(* IEC 61131-3 sources: beckhoffAutomationInterface/ST/Shark/Lib/BehaviorTree/actions, 12 files *)

(* ---- FB_AlwaysFailureNode.st ---- *)
FUNCTION_BLOCK FB_AlwaysFailureNode IMPLEMENTS I_TreeNode
VAR_INPUT
    sName : STRING(50) := 'Always Failure';
END_VAR

METHOD Tick : ST_NodeResult
    Tick.eStatus := E_NodeStatus.FAILURE;
    Tick.bHasError := TRUE;
    Tick.stError.eErrorId := E_ErrorId.ERR_BT_FORCED_FAILURE;
    Tick.stError.sSource := sName;
    Tick.stError.sMessage := 'Forced Failure';
    Tick.sDescription := CONCAT(sName, ' - Failure');
END_METHOD

{attribute 'estimated-stack-usage' := '500'}
METHOD Reset : BOOL
    Reset := TRUE;
END_METHOD

{attribute 'estimated-stack-usage' := '500'}
METHOD Halt
END_METHOD
END_FUNCTION_BLOCK

(* ---- FB_AlwaysSuccessNode.st ---- *)
FUNCTION_BLOCK FB_AlwaysSuccessNode IMPLEMENTS I_TreeNode
VAR_INPUT
    sName : STRING(50) := 'Always Success';
END_VAR

METHOD Tick : ST_NodeResult
    Tick.eStatus := E_NodeStatus.SUCCESS;
    Tick.rProgress := 100.0;
    Tick.sDescription := CONCAT(sName, ' - Success');
END_METHOD

{attribute 'estimated-stack-usage' := '500'}
METHOD Reset : BOOL
    Reset := TRUE;
END_METHOD

{attribute 'estimated-stack-usage' := '500'}
METHOD Halt
END_METHOD
END_FUNCTION_BLOCK

(* ---- FB_CheckSensorNode.st ---- *)
FUNCTION_BLOCK FB_CheckSensorNode IMPLEMENTS I_TreeNode
VAR_INPUT
    sName : STRING(50) := 'Check Sensor Node';
END_VAR
VAR
    _ipSensor     : I_Sensor;
    _rThreshold   : LREAL;
    _eCompareMode : E_CompareMode := E_CompareMode.GREATER_THAN;
    _rTolerance   : LREAL;
    _rLastValue   : LREAL;
END_VAR

METHOD PUBLIC Init : BOOL
VAR_INPUT
    ipSensor   : I_Sensor;
    rThreshold : LREAL;
    eMode      : E_CompareMode := E_CompareMode.GREATER_THAN;
    rTolerance : LREAL := 0.0;
    sNodeName  : STRING(50) := '';
END_VAR
    IF ipSensor = 0 THEN RETURN; END_IF
    _ipSensor     := ipSensor;
    _rThreshold   := rThreshold;
    _eCompareMode := eMode;
    _rTolerance   := rTolerance;
    IF sNodeName <> '' THEN sName := sNodeName; END_IF
    Init := TRUE;
END_METHOD

PROPERTY PUBLIC Threshold : LREAL
    GET
    Threshold := _rThreshold;
    END_GET
    SET
    _rThreshold := Threshold;
    END_SET
END_PROPERTY

PROPERTY PUBLIC CompareMode : E_CompareMode
    GET
    CompareMode := _eCompareMode;
    END_GET
    SET
    _eCompareMode := CompareMode;
    END_SET
END_PROPERTY

METHOD PRIVATE GetStatusDescription : STRING(255)
VAR
    sResult : STRING(255);
END_VAR
    sResult := CONCAT(sName, ' - current=');
    sResult := CONCAT(sResult, LREAL_TO_FMTSTR(_rLastValue, 2, TRUE));
    sResult := CONCAT(sResult, CONCAT(', threshold=', LREAL_TO_FMTSTR(_rThreshold, 2, TRUE)));
    IF _eCompareMode = E_CompareMode.WITHIN_TOLERANCE AND _rTolerance > 0.0 THEN
        sResult := CONCAT(sResult, CONCAT(' +/-', LREAL_TO_FMTSTR(_rTolerance, 2, TRUE)));
    ELSE
        sResult := CONCAT(sResult, CONCAT(' (', CONCAT(F_CompareModeToString(_eCompareMode), ')')));
    END_IF
    GetStatusDescription := sResult;
END_METHOD

METHOD Tick : ST_NodeResult
VAR
    rCurrent  : LREAL;
    sErrorMsg : STRING(255);
END_VAR
    IF _ipSensor = 0 THEN
        Tick := F_BuildNullInterfaceResult(sName, 'Sensor interface not configured');
        RETURN;
    END_IF

    IF _ipSensor.IsError() THEN
        Tick.eStatus := E_NodeStatus.FAILURE;
        Tick.bHasError := TRUE;
        Tick.stError.eErrorId := E_ErrorId.ERR_BT_SENSOR_ERROR;
        Tick.stError.sSource := sName;
        Tick.stError.sMessage := 'Sensor reported error';
        RETURN;
    END_IF

    rCurrent    := _ipSensor.GetMeasurement();
    _rLastValue := rCurrent;

    IF F_EvaluateCompareMode(rCurrent, _rThreshold, _rTolerance, _eCompareMode) THEN
        Tick.eStatus := E_NodeStatus.SUCCESS;
        Tick.rProgress := 100.0;
        Tick.sDescription := GetStatusDescription();
    ELSE
        sErrorMsg := CONCAT('Value ', LREAL_TO_FMTSTR(rCurrent, 2, TRUE));
        sErrorMsg := CONCAT(sErrorMsg, CONCAT(' not ', F_CompareModeToString(_eCompareMode)));
        sErrorMsg := CONCAT(sErrorMsg, CONCAT(' ', LREAL_TO_FMTSTR(_rThreshold, 2, TRUE)));

        Tick.eStatus := E_NodeStatus.FAILURE;
        Tick.bHasError := TRUE;
        Tick.stError.eErrorId := E_ErrorId.ERR_BT_CONDITION_FAILED;
        Tick.stError.sSource := sName;
        Tick.stError.sMessage := sErrorMsg;
        Tick.sDescription := GetStatusDescription();
    END_IF
END_METHOD

{attribute 'estimated-stack-usage' := '500'}
METHOD Halt
    // No explicit action required
END_METHOD

{attribute 'estimated-stack-usage' := '500'}
METHOD Reset : BOOL
    Reset := TRUE;
END_METHOD

END_FUNCTION_BLOCK

(* ---- FB_CloseValveNode.st ---- *)
FUNCTION_BLOCK FB_CloseValveNode IMPLEMENTS I_TreeNode
VAR_INPUT
    sName : STRING(50) := 'Close Valve';
END_VAR
VAR
    _ipValve : I_Valve;
END_VAR

METHOD PUBLIC Init : BOOL
VAR_INPUT
    ipValve   : I_Valve;
    sNodeName : STRING(50) := '';
END_VAR
    IF ipValve = 0 THEN RETURN; END_IF
    _ipValve := ipValve;
    IF sNodeName <> '' THEN sName := sNodeName; END_IF
    Init := TRUE;
END_METHOD

METHOD Tick : ST_NodeResult
VAR
    stValveError : ST_Error;
END_VAR
    IF _ipValve = 0 THEN
        Tick := F_BuildNullInterfaceResult(sName, 'Valve interface not configured');
        RETURN;
    END_IF

    _ipValve.Close();

    IF _ipValve.IsClosed() THEN
        Tick.eStatus := E_NodeStatus.SUCCESS;
        Tick.rProgress := 100.0;
        Tick.sDescription := CONCAT(sName, ' - Valve closed');
    ELSIF _ipValve.IsError() THEN
        stValveError := _ipValve.GetError();
        Tick.eStatus := E_NodeStatus.FAILURE;
        Tick.bHasError := TRUE;
        Tick.stError.sSource := sName;

        IF stValveError.eErrorId <> E_ErrorId.NO_ERROR THEN
            Tick.stError.eErrorId := stValveError.eErrorId;
            Tick.stError.sMessage := stValveError.sMessage;
        ELSE
            Tick.stError.eErrorId := E_ErrorId.ERR_BT_VALVE_ERROR;
            Tick.stError.sMessage := 'Valve reported error while closing';
        END_IF
    ELSE
        Tick.eStatus := E_NodeStatus.RUNNING;
        Tick.sDescription := CONCAT(sName, ' - Closing valve, currently open');
    END_IF
END_METHOD

{attribute 'estimated-stack-usage' := '500'}
METHOD Reset : BOOL
    Reset := TRUE;
END_METHOD

{attribute 'estimated-stack-usage' := '500'}
METHOD Halt
    // Safe state: ensure the valve is closed (isolated).
    IF _ipValve <> 0 THEN
        _ipValve.Close();
    END_IF
END_METHOD

END_FUNCTION_BLOCK

(* ---- FB_ConditionNode.st ---- *)
// FB_ConditionNode - Pure leaf node that evaluates a boolean condition
// Returns SUCCESS if condition is TRUE, FAILURE if FALSE
// This is a leaf node, it has no child.
//
// Usage:
//   fbCondition.Init(refCondition := bMyFlag);
//   fbSequence.AddChild(fbCondition);
//
FUNCTION_BLOCK FB_ConditionNode IMPLEMENTS I_TreeNode
VAR_INPUT
    sName : STRING(50) := 'Condition Node';
END_VAR
VAR
    _refCondition : REFERENCE TO BOOL;
    _bInvertResult : BOOL := FALSE;
END_VAR

    // Configure with reference to boolean condition
METHOD PUBLIC Init : BOOL
VAR_INPUT
    refCondition  : REFERENCE TO BOOL;
    bInvertResult : BOOL := FALSE; // Optional: invert the result
    sNodeName     : STRING(50) := '';
END_VAR
    IF NOT __ISVALIDREF(refCondition) THEN
        Init := FALSE;
        RETURN;
    END_IF

    _refCondition REF= refCondition;
    _bInvertResult := bInvertResult;
    IF sNodeName <> '' THEN sName := sNodeName; END_IF
    Init := TRUE;
END_METHOD

METHOD Tick : ST_NodeResult
VAR
    bConditionValue : BOOL;
END_VAR

    IF NOT __ISVALIDREF(_refCondition) THEN
        Tick.eStatus := E_NodeStatus.FAILURE;
        Tick.bHasError := TRUE;
        Tick.stError.eErrorId := E_ErrorId.ERR_BT_CONDITION_NOT_CONFIGURED;
        Tick.stError.sSource := sName;
        Tick.stError.sMessage := 'Condition reference not configured';
        RETURN;
    END_IF

    bConditionValue := _refCondition;

    // Apply inversion if configured
    IF _bInvertResult THEN
        bConditionValue := NOT bConditionValue;
    END_IF

    IF bConditionValue THEN
        Tick.eStatus := E_NodeStatus.SUCCESS;
        Tick.sDescription := CONCAT(sName, ' - Condition Met');
        Tick.rProgress := 100.0;
    ELSE
        // Condition false is not an error - it's expected behavior
        Tick.eStatus := E_NodeStatus.FAILURE;
        Tick.sDescription := CONCAT(sName, ' - Condition Not Met');
    END_IF
END_METHOD

{attribute 'estimated-stack-usage' := '500'}
METHOD Halt
    // Nothing to halt
END_METHOD

{attribute 'estimated-stack-usage' := '500'}
METHOD Reset : BOOL
    Reset := TRUE;
END_METHOD

END_FUNCTION_BLOCK

(* ---- FB_EnableControllerNode.st ---- *)
FUNCTION_BLOCK FB_EnableControllerNode IMPLEMENTS I_TreeNode
VAR_INPUT
    sName : STRING(50) := 'Enable Controller';
END_VAR
VAR
    _ipController : I_Controller;
    _bEnable      : BOOL;
END_VAR

METHOD PUBLIC Init : BOOL
VAR_INPUT
    ipController : I_Controller;
    bEnable      : BOOL;
    sNodeName    : STRING(50) := '';
END_VAR
    IF ipController = 0 THEN RETURN; END_IF
    _ipController := ipController;
    _bEnable      := bEnable;
    IF sNodeName <> '' THEN sName := sNodeName; END_IF
    Init := TRUE;
END_METHOD

METHOD Tick : ST_NodeResult
    IF _ipController = 0 THEN
        Tick := F_BuildNullInterfaceResult(sName, 'Controller interface not configured');
        RETURN;
    END_IF

    _ipController.Enable(_bEnable);
    Tick.eStatus := E_NodeStatus.SUCCESS;
    Tick.rProgress := 100.0;
    IF _bEnable THEN
        Tick.sDescription := CONCAT(sName, ' - Enabling controller');
    ELSE
        Tick.sDescription := CONCAT(sName, ' - Disabling controller');
    END_IF
END_METHOD

{attribute 'estimated-stack-usage' := '500'}
METHOD Reset : BOOL
    Reset := TRUE;
END_METHOD

{attribute 'estimated-stack-usage' := '500'}
METHOD Halt
    // Safe state: disable the controller.
    IF _ipController <> 0 THEN
        _ipController.Enable(FALSE);
    END_IF
END_METHOD

END_FUNCTION_BLOCK

(* ---- FB_MonitorControllerNode.st ---- *)
(* FB_MonitorControllerNode - Monitor controller for errors while running

BEHAVIOR:
- Returns RUNNING while controller has no error
- Returns FAILURE immediately if controller reports error
- Never returns SUCCESS on its own (used in parallel with other nodes)

USE CASE:
Run in parallel with other nodes. If the controller enters an error state
this node fails immediately, causing the parallel node to fail without
waiting for the other branches to complete.
*)
FUNCTION_BLOCK FB_MonitorControllerNode IMPLEMENTS I_TreeNode
VAR_INPUT
    sName : STRING(50) := 'Monitor Controller Node';
END_VAR
VAR
    _ipController : I_Controller;
END_VAR

METHOD PUBLIC Init : BOOL
VAR_INPUT
    ipController : I_Controller;
    sNodeName    : STRING(50) := '';
END_VAR
    IF ipController = 0 THEN RETURN; END_IF
    _ipController := ipController;
    IF sNodeName <> '' THEN sName := sNodeName; END_IF
    Init := TRUE;
END_METHOD

METHOD Tick : ST_NodeResult
VAR
    stStatus : ST_ControllerStatus;
END_VAR
    IF _ipController = 0 THEN
        Tick := F_BuildNullInterfaceResult(sName, 'Controller interface not configured');
        RETURN;
    END_IF

    stStatus := _ipController.GetStatus();
    IF stStatus.stError.eErrorId <> E_ErrorId.NO_ERROR THEN
        Tick.eStatus := E_NodeStatus.FAILURE;
        Tick.bHasError := TRUE;
        Tick.stError := stStatus.stError;
        RETURN;
    END_IF

    Tick.eStatus := E_NodeStatus.RUNNING;
    Tick.sDescription := CONCAT(sName, ' - Monitoring (OK)');
END_METHOD

{attribute 'estimated-stack-usage' := '500'}
METHOD Halt
    // No explicit action required
END_METHOD

{attribute 'estimated-stack-usage' := '500'}
METHOD Reset : BOOL
    Reset := TRUE;
END_METHOD

END_FUNCTION_BLOCK

(* ---- FB_OpenValveNode.st ---- *)
FUNCTION_BLOCK FB_OpenValveNode IMPLEMENTS I_TreeNode
VAR_INPUT
    sName : STRING(50) := 'Open Valve';
END_VAR
VAR
    _ipValve : I_Valve;
END_VAR

METHOD PUBLIC Init : BOOL
VAR_INPUT
    ipValve   : I_Valve;
    sNodeName : STRING(50) := '';
END_VAR
    IF ipValve = 0 THEN RETURN; END_IF
    _ipValve := ipValve;
    IF sNodeName <> '' THEN sName := sNodeName; END_IF
    Init := TRUE;
END_METHOD

METHOD Tick : ST_NodeResult
VAR
    stValveError : ST_Error;
END_VAR
    IF _ipValve = 0 THEN
        Tick := F_BuildNullInterfaceResult(sName, 'Valve interface not configured');
        RETURN;
    END_IF

    _ipValve.Open();

    IF _ipValve.IsOpen() THEN
        Tick.eStatus := E_NodeStatus.SUCCESS;
        Tick.rProgress := 100.0;
        Tick.sDescription := CONCAT(sName, ' - Valve open');
    ELSIF _ipValve.IsError() THEN
        stValveError := _ipValve.GetError();
        Tick.eStatus := E_NodeStatus.FAILURE;
        Tick.bHasError := TRUE;
        Tick.stError.sSource := sName;

        IF stValveError.eErrorId <> E_ErrorId.NO_ERROR THEN
            Tick.stError.eErrorId := stValveError.eErrorId;
            Tick.stError.sMessage := stValveError.sMessage;
        ELSE
            Tick.stError.eErrorId := E_ErrorId.ERR_BT_VALVE_ERROR;
            Tick.stError.sMessage := 'Valve reported error while opening';
        END_IF
    ELSE
        Tick.eStatus := E_NodeStatus.RUNNING;
        Tick.sDescription := CONCAT(sName, ' - Opening valve, currently closed');
    END_IF
END_METHOD

{attribute 'estimated-stack-usage' := '500'}
METHOD Reset : BOOL
    Reset := TRUE;
END_METHOD

{attribute 'estimated-stack-usage' := '500'}
METHOD Halt
    // Safe state: isolate by closing the valve (SEQUENCE_BT_LIFECYCLE.md §3).
    IF _ipValve <> 0 THEN
        _ipValve.Close();
    END_IF
END_METHOD

END_FUNCTION_BLOCK

(* ---- FB_SetControllerNode.st ---- *)
FUNCTION_BLOCK FB_SetControllerNode IMPLEMENTS I_TreeNode
VAR_INPUT
    sName : STRING(50) := 'Set Controller';
END_VAR
VAR
    _ipController : I_Controller;
    _rSetpoint    : LREAL;
END_VAR

METHOD PUBLIC Init : BOOL
VAR_INPUT
    ipController : I_Controller;
    rSetpoint    : LREAL;
    sNodeName    : STRING(50) := '';
END_VAR
    IF ipController = 0 THEN RETURN; END_IF
    _ipController := ipController;
    _rSetpoint    := rSetpoint;
    IF sNodeName <> '' THEN sName := sNodeName; END_IF
    Init := TRUE;
END_METHOD

PROPERTY PUBLIC Setpoint : LREAL
    GET
    Setpoint := _rSetpoint;
    END_GET
    SET
    _rSetpoint := Setpoint;
    END_SET
END_PROPERTY

METHOD Tick : ST_NodeResult
    IF _ipController = 0 THEN
        Tick := F_BuildNullInterfaceResult(sName, 'Controller interface not configured');
        RETURN;
    END_IF

    _ipController.SetSetpoint(_rSetpoint);
    Tick.eStatus := E_NodeStatus.SUCCESS;
    Tick.rProgress := 100.0;
    Tick.sDescription := CONCAT(sName, CONCAT(' - Set setpoint=', LREAL_TO_FMTSTR(_rSetpoint, 2, TRUE)));
END_METHOD

{attribute 'estimated-stack-usage' := '500'}
METHOD Reset : BOOL
    Reset := TRUE;
END_METHOD

{attribute 'estimated-stack-usage' := '500'}
METHOD Halt
    // Safe state: zero the setpoint.
    IF _ipController <> 0 THEN
        _ipController.SetSetpoint(0.0);
    END_IF
END_METHOD

END_FUNCTION_BLOCK

(* ---- FB_SetDigitalOutputNode.st ---- *)
FUNCTION_BLOCK FB_SetDigitalOutputNode IMPLEMENTS I_TreeNode
VAR_INPUT
    sName : STRING(50) := 'Set Digital Output Node';
END_VAR
VAR
    _ipDO : I_DigitalOutput;
    _bState : BOOL;
END_VAR

METHOD PUBLIC Init : BOOL
VAR_INPUT
    ipDO      : I_DigitalOutput;
    bState    : BOOL;
    sNodeName : STRING(50) := '';
END_VAR
    IF ipDO = 0 THEN RETURN; END_IF
    _ipDO   := ipDO;
    _bState := bState;
    IF sNodeName <> '' THEN sName := sNodeName; END_IF
    Init := TRUE;
END_METHOD

METHOD Tick : ST_NodeResult
    IF _ipDO = 0 THEN
        Tick := F_BuildNullInterfaceResult(sName, 'Digital output interface not configured');
        RETURN;
    END_IF

    _ipDO.SetOutput(_bState);
    Tick.eStatus := E_NodeStatus.SUCCESS;
    Tick.sDescription := CONCAT(sName, ' - Output set');
    Tick.rProgress := 100.0;
END_METHOD

{attribute 'estimated-stack-usage' := '500'}
METHOD Halt
    // Apply the safe state configured at Init time.
    // The node has no knowledge of whether safe means TRUE or FALSE.
    IF _ipDO <> 0 THEN
        _ipDO.SetSafeState();
    END_IF
END_METHOD

{attribute 'estimated-stack-usage' := '500'}
METHOD Reset : BOOL
    Reset := TRUE;
END_METHOD

END_FUNCTION_BLOCK

(* ---- FB_WaitForSensorNode.st ---- *)
(* FB_WaitForSensorNode - Wait until sensor meets a condition

BEHAVIOR:
- Returns RUNNING while waiting for condition
- Returns SUCCESS when condition is met
- Returns FAILURE on errors (null sensor, sensor error) or timeout

TIMEOUT:
- tTimeout = T#0S  => no timeout, wait indefinitely (default)
- tTimeout > T#0S  => FAILURE with descriptive message when timeout expires

COMPARE MODES:
- WITHIN_TOLERANCE: ABS(value - target) <= tolerance (default)
- GREATER_THAN:     value > target
- LESS_THAN:        value < target
*)
FUNCTION_BLOCK FB_WaitForSensorNode IMPLEMENTS I_TreeNode
VAR_INPUT
    sName : STRING(50) := 'Wait For Sensor Node';
END_VAR
VAR
    _ipSensor     : I_Sensor;
    _rTarget      : LREAL;
    _rTolerance   : LREAL;
    _eCompareMode : E_CompareMode := E_CompareMode.WITHIN_TOLERANCE;
    _rLastValue   : LREAL;
    _tTimeout     : TIME := T#0S;
    _fbTimer      : TON;
    _bStarted     : BOOL;
END_VAR

METHOD PUBLIC Init : BOOL
VAR_INPUT
    ipSensor   : I_Sensor;
    rTarget    : LREAL;
    rTolerance : LREAL := 0.0;
    eMode      : E_CompareMode := E_CompareMode.WITHIN_TOLERANCE;
    tTimeout   : TIME := T#0S;
    sNodeName  : STRING(50) := '';
END_VAR
    IF ipSensor = 0 THEN RETURN; END_IF
    _ipSensor     := ipSensor;
    _rTarget      := rTarget;
    _rTolerance   := rTolerance;
    _eCompareMode := eMode;
    _tTimeout     := tTimeout;
    IF sNodeName <> '' THEN sName := sNodeName; END_IF
    Init := TRUE;
END_METHOD

PROPERTY PUBLIC Target : LREAL
    GET
    Target := _rTarget;
    END_GET
    SET
    _rTarget := Target;
    END_SET
END_PROPERTY

PROPERTY PUBLIC Tolerance : LREAL
    GET
    Tolerance := _rTolerance;
    END_GET
    SET
    _rTolerance := Tolerance;
    END_SET
END_PROPERTY

PROPERTY PUBLIC CompareMode : E_CompareMode
    GET
    CompareMode := _eCompareMode;
    END_GET
    SET
    _eCompareMode := CompareMode;
    END_SET
END_PROPERTY

PROPERTY PUBLIC Timeout : TIME
    GET
    Timeout := _tTimeout;
    END_GET
    SET
    _tTimeout := Timeout;
    END_SET
END_PROPERTY

METHOD PUBLIC GetStatusDescription : STRING(255)
VAR
    sResult : STRING(255);
END_VAR
    sResult := CONCAT(sName, ' - current=');
    sResult := CONCAT(sResult, LREAL_TO_FMTSTR(_rLastValue, 2, TRUE));
    sResult := CONCAT(sResult, CONCAT(', target=', LREAL_TO_FMTSTR(_rTarget, 2, TRUE)));
    IF _eCompareMode = E_CompareMode.WITHIN_TOLERANCE AND _rTolerance > 0.0 THEN
        sResult := CONCAT(sResult, CONCAT(' +/-', LREAL_TO_FMTSTR(_rTolerance, 2, TRUE)));
    ELSE
        sResult := CONCAT(sResult, CONCAT(' (', CONCAT(F_CompareModeToString(_eCompareMode), ')')));
    END_IF
    IF _tTimeout > T#0S AND _bStarted THEN
        sResult := CONCAT(sResult, CONCAT(' timeout=', CONCAT(TIME_TO_STRING(_fbTimer.ET), CONCAT('/', TIME_TO_STRING(_tTimeout)))));
    END_IF
    GetStatusDescription := sResult;
END_METHOD

METHOD Tick : ST_NodeResult
VAR
    rCurrentVal : LREAL;
END_VAR
    IF _ipSensor = 0 THEN
        Tick := F_BuildNullInterfaceResult(sName, 'Sensor interface not configured');
        RETURN;
    END_IF

    IF _ipSensor.IsError() THEN
        Tick.eStatus := E_NodeStatus.FAILURE;
        Tick.bHasError := TRUE;
        Tick.stError.eErrorId := E_ErrorId.ERR_BT_SENSOR_ERROR;
        Tick.stError.sSource := sName;
        Tick.stError.sMessage := 'Sensor reported error';
        RETURN;
    END_IF

    IF NOT _bStarted THEN
        _bStarted := TRUE;
    END_IF

    IF _tTimeout > T#0S THEN
        _fbTimer(IN := _bStarted, PT := _tTimeout);
        IF _fbTimer.Q THEN
            Tick.eStatus := E_NodeStatus.FAILURE;
            Tick.bHasError := TRUE;
            Tick.stError.eErrorId := E_ErrorId.ERR_BT_TIMEOUT;
            Tick.stError.sSource := sName;
            Tick.stError.sMessage := CONCAT(
                    CONCAT('Timeout after ', TIME_TO_STRING(_tTimeout)),
                    CONCAT(' - current=', CONCAT(LREAL_TO_FMTSTR(_rLastValue, 2, TRUE), CONCAT(', target=', LREAL_TO_FMTSTR(_rTarget, 2, TRUE))))
                );
            RETURN;
        END_IF
        Tick.rProgress := (TIME_TO_REAL(_fbTimer.ET) / TIME_TO_REAL(_tTimeout)) * 100.0;
        IF Tick.rProgress > 100.0 THEN Tick.rProgress := 100.0; END_IF
    END_IF

    rCurrentVal := _ipSensor.GetMeasurement();
    _rLastValue := rCurrentVal;

    IF F_EvaluateCompareMode(rCurrentVal, _rTarget, _rTolerance, _eCompareMode) THEN
        _bStarted := FALSE;
        _fbTimer(IN := FALSE);

        Tick.eStatus := E_NodeStatus.SUCCESS;
        Tick.rProgress := 100.0;
        Tick.sDescription := GetStatusDescription();
    ELSE
        Tick.eStatus := E_NodeStatus.RUNNING;
        Tick.sDescription := GetStatusDescription();
    END_IF

END_METHOD

{attribute 'estimated-stack-usage' := '500'}
METHOD Halt
    // Stop timers, preserve state
    _bStarted := FALSE;
    _fbTimer(IN := FALSE);
END_METHOD

{attribute 'estimated-stack-usage' := '500'}
METHOD Reset : BOOL
    _bStarted := FALSE;
    _fbTimer(IN := FALSE);
    Reset := TRUE;
END_METHOD

END_FUNCTION_BLOCK

(* ---- FB_WaitNode.st ---- *)
FUNCTION_BLOCK FB_WaitNode IMPLEMENTS I_TreeNode
VAR_INPUT
    sName : STRING(50) := 'Wait';
END_VAR
VAR
    _tWaitTime : TIME := T#2S;
    _fbTimer : TON;
    _bStarted : BOOL := FALSE;
END_VAR

METHOD PUBLIC Init : BOOL
VAR_INPUT
    tWaitTime : TIME;
    sNodeName : STRING(50) := '';
END_VAR
    _tWaitTime := tWaitTime;
    IF sNodeName <> '' THEN sName := sNodeName; END_IF
    Init := TRUE;
END_METHOD

// Property to get/set wait time at runtime
PROPERTY PUBLIC WaitTime : TIME
    GET
    WaitTime := _tWaitTime;
    END_GET
    SET
    _tWaitTime := WaitTime;
    END_SET
END_PROPERTY

METHOD Tick : ST_NodeResult
    // Call timer unconditionally every scan cycle
    _fbTimer(IN := _bStarted, PT := _tWaitTime);

    IF NOT _bStarted THEN
        _bStarted := TRUE;
        Tick.eStatus := E_NodeStatus.RUNNING;
        Tick.rProgress := 0.0;
        Tick.bHasError := FALSE;
        Tick.sDescription := CONCAT(sName, CONCAT(' - Wait ', TIME_TO_STRING(_tWaitTime)));
        RETURN;
    END_IF

    // Calculate progress based on elapsed time
    IF _tWaitTime > T#0S THEN
        Tick.rProgress := (TIME_TO_REAL(_fbTimer.ET) / TIME_TO_REAL(_tWaitTime)) * 100.0;
        IF Tick.rProgress > 100.0 THEN Tick.rProgress := 100.0; END_IF
    ELSE
        Tick.rProgress := 100.0;
    END_IF

    IF _fbTimer.Q THEN
        _bStarted := FALSE; // Reset for next full execution
        Tick.eStatus := E_NodeStatus.SUCCESS;
        Tick.rProgress := 100.0;
        Tick.sDescription := CONCAT(sName, ' - Done');
    ELSE
        Tick.eStatus := E_NodeStatus.RUNNING;
        Tick.sDescription := CONCAT(sName, CONCAT(' - Waiting ', CONCAT(TIME_TO_STRING(_fbTimer.ET), CONCAT('/', TIME_TO_STRING(_tWaitTime)))));
    END_IF
END_METHOD

    // Method: Halt - Stops execution but preserves error state
{attribute 'estimated-stack-usage' := '500'}
METHOD Halt
    _bStarted := FALSE;
    _fbTimer(IN := FALSE);
END_METHOD

{attribute 'estimated-stack-usage' := '500'}
METHOD Reset : BOOL
    _bStarted := FALSE;
    _fbTimer(IN := FALSE);
    Reset := TRUE;
END_METHOD

END_FUNCTION_BLOCK
